{attribute 'hide_all_locals'}
FUNCTION_BLOCK ResetGroup EXTENDS TaskBase
VAR_INPUT
END_VAR
VAR_OUTPUT
END_VAR
VAR
	groupReset			: MC_GroupReset;
	_caGroup			: ICollisionGroup;
	_resetGroup : BOOL;
	Logger : TcMessage_Ext;
END_VAR

{analysis -2}

METHOD Abort : BOOL
groupReset.Execute := FALSE;
State := 0;
Abort := true;
END_METHOD

METHOD Cycle : HRESULT
VAR_INPUT
END_VAR
CASE State OF
	0:
		IF _resetGroup THEN
			Cycle := S_PENDING;
			_Done := FALSE;
			_Error := FALSE;
			_Busy := TRUE;
			groupReset.Execute := TRUE;
			IF groupReset.Busy THEN
				State := 10;
				_resetGroup := FALSE;
				Logger.Send(TC_EVENTS.XtsCaGroupEvents.CAGroupResetting,'');
			END_IF
		END_IF
	
	10:
		IF NOT groupReset.Busy THEN
			IF groupReset.Done THEN
				_Done := TRUE;
				Logger.Send(TC_EVENTS.XtsCaGroupEvents.CAGroupResetDone,'');
			ELSIF groupReset.Error THEN
				_Error := TRUE;
				Logger.Send(TC_EVENTS.XtsCaGroupEvents.CAGroupResetError,'');
			END_IF
			_Busy := FALSE;
			groupReset.Execute := false;
			State := 0;
			Cycle := S_OK;
		END_IF
END_CASE


groupReset(AxesGroup := _caGroup.GroupRef);
END_METHOD

METHOD Execute : BOOL
Execute := _resetGroup := true;
END_METHOD

METHOD FB_init : BOOL
VAR_INPUT
	bInitRetains : BOOL; // if TRUE, the retain variables are initialized (warm start / cold start)
	bInCopyCode : BOOL;  // if TRUE, the instance afterwards gets moved into the copy code (online change)
	MyCaGroup : ICollisionGroup;	
END_VAR
_caGroup := MyCaGroup;
END_METHOD

END_FUNCTION_BLOCK

(* stored: Version 1.1.0.1, ProductVersion 3.1.4024.12
   POU ResetGroup: Id {c0d0b360-5fec-467e-a65e-491de04b13b3}, SpecialFunc None
   Method Abort: Id {713891a3-4780-46dc-94db-48974077b800}
   Method Cycle: Id {60490ba9-dc4f-4168-a59d-a16c9df8b6fb}
   Method Execute: Id {d2d6e3c9-1d94-473e-8bef-e969b6fceb58}
   Method FB_init: Id {747a23bd-39e4-4843-a82d-196c2af18fd6} *)
